// TIA Portal V20 export
FUNCTION_BLOCK "F-FB_DigitalInput"   // FB110, F_LAD
{ S7_Optimized_Access := 'TRUE' }
// stored: AutoNumber false
   VAR
      sSafety_EStop : EV1oo2DI;
      sKeySettingMode : EV1oo2DI;
      sKeySettingLaser : EV1oo2DI;
      sMaintenanceDoorClosed : EV1oo2DI;
      sFrontDoorClosed : EV1oo2DI;
      sEmergencyStopPowerLaser : EV1oo2DI;
      sRoofLeftDoorClosed : EV1oo2DI;
      sKeyLaserON : EV1oo2DI;
      sLaserExternDoorClosed : EV1oo2DI;
      sSasOneDoorClosed : EV1oo2DI;
      sBwLoaderDoorClosed : EV1oo2DI;
      sRoofRightDoorClosed : EV1oo2DI;
      sSonplas_EStop : EV1oo2DI;
      sBwLoader_EStop : EV1oo2DI;
      sSonplasDoorClosed : EV1oo2DI;
      sAck_iSafety_EStop { ExternalAccessible := 'False'; ExternalVisible := 'False'; ExternalWritable := 'False'} : Bool;
      sAck_iKeySettingMode { ExternalAccessible := 'False'; ExternalVisible := 'False'; ExternalWritable := 'False'} : Bool;
      sAck_iKeySettingLaser { ExternalAccessible := 'False'; ExternalVisible := 'False'; ExternalWritable := 'False'} : Bool;
      sAck_iMaintenanceDoorClosed { ExternalAccessible := 'False'; ExternalVisible := 'False'; ExternalWritable := 'False'} : Bool;
      sAck_iFrontDoorClosed { ExternalAccessible := 'False'; ExternalVisible := 'False'; ExternalWritable := 'False'} : Bool;
      sAck_iEmergencyStopPowerLaser { ExternalAccessible := 'False'; ExternalVisible := 'False'; ExternalWritable := 'False'} : Bool;
      sAck_iRoofLeftDoorClosed { ExternalAccessible := 'False'; ExternalVisible := 'False'; ExternalWritable := 'False'} : Bool;
      sAck_iKeyLaserON { ExternalAccessible := 'False'; ExternalVisible := 'False'; ExternalWritable := 'False'} : Bool;
      sAck_iLaserExternDoorClosed : Bool;
      sAck_iSasOneDoorClosed { ExternalAccessible := 'False'; ExternalVisible := 'False'; ExternalWritable := 'False'} : Bool;
      sAck_iBwLoaderDoorClosed : Bool;
      sAck_iRoofRightDoorClosed { ExternalAccessible := 'False'; ExternalVisible := 'False'; ExternalWritable := 'False'} : Bool;
      sAck_iSonplas_EStop : Bool;
      sAck_iBwLoader_EStop : Bool;
      sAck_iSonplasDoorClosed { ExternalAccessible := 'False'; ExternalVisible := 'False'; ExternalWritable := 'False'} : Bool;
   END_VAR
BEGIN

REGION Network 1: Safety EStop
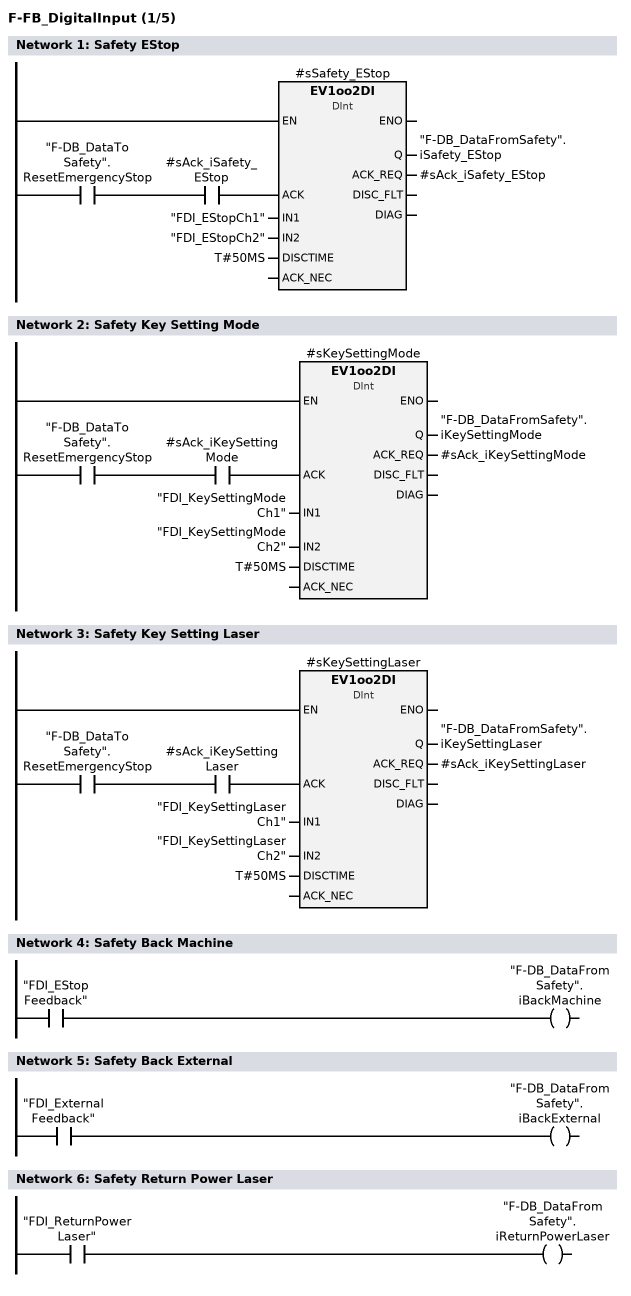
   RUNG wire#powerrail
      { S7_Templates := "codedbool_type := DInt" } #sSafety_EStop.EV1oo2DI(ACK := wire#w1, IN1 := "FDI_EStopCh1", IN2 := "FDI_EStopCh2", DISCTIME := T#50MS, ACK_NEC :=, Q => "F-DB_DataFromSafety".iSafety_EStop, ACK_REQ => #sAck_iSafety_EStop, DISC_FLT =>, DIAG =>)
   END_RUNG
   RUNG wire#powerrail
      Contact( "F-DB_DataToSafety".ResetEmergencyStop )
      Contact( #sAck_iSafety_EStop )
   END_RUNG wire#w1
   // the same network as SCL:
   #sSafety_EStop(ACK := "F-DB_DataToSafety".ResetEmergencyStop AND #sAck_iSafety_EStop,   // EV1oo2DI
                  IN1 := "FDI_EStopCh1",
                  IN2 := "FDI_EStopCh2",
                  DISCTIME := T#50MS,
                  Q => "F-DB_DataFromSafety".iSafety_EStop,
                  ACK_REQ => #sAck_iSafety_EStop);
END_REGION

REGION Network 2: Safety Key Setting Mode
   RUNG wire#powerrail
      { S7_Templates := "codedbool_type := DInt" } #sKeySettingMode.EV1oo2DI(ACK := wire#w1, IN1 := "FDI_KeySettingModeCh1", IN2 := "FDI_KeySettingModeCh2", DISCTIME := T#50MS, ACK_NEC :=, Q => "F-DB_DataFromSafety".iKeySettingMode, ACK_REQ => #sAck_iKeySettingMode, DISC_FLT =>, DIAG =>)
   END_RUNG
   RUNG wire#powerrail
      Contact( "F-DB_DataToSafety".ResetEmergencyStop )
      Contact( #sAck_iKeySettingMode )
   END_RUNG wire#w1
   // the same network as SCL:
   #sKeySettingMode(ACK := "F-DB_DataToSafety".ResetEmergencyStop AND #sAck_iKeySettingMode,   // EV1oo2DI
                    IN1 := "FDI_KeySettingModeCh1",
                    IN2 := "FDI_KeySettingModeCh2",
                    DISCTIME := T#50MS,
                    Q => "F-DB_DataFromSafety".iKeySettingMode,
                    ACK_REQ => #sAck_iKeySettingMode);
END_REGION

REGION Network 3: Safety Key Setting Laser
   RUNG wire#powerrail
      { S7_Templates := "codedbool_type := DInt" } #sKeySettingLaser.EV1oo2DI(ACK := wire#w1, IN1 := "FDI_KeySettingLaserCh1", IN2 := "FDI_KeySettingLaserCh2", DISCTIME := T#50MS, ACK_NEC :=, Q => "F-DB_DataFromSafety".iKeySettingLaser, ACK_REQ => #sAck_iKeySettingLaser, DISC_FLT =>, DIAG =>)
   END_RUNG
   RUNG wire#powerrail
      Contact( "F-DB_DataToSafety".ResetEmergencyStop )
      Contact( #sAck_iKeySettingLaser )
   END_RUNG wire#w1
   // the same network as SCL:
   #sKeySettingLaser(ACK := "F-DB_DataToSafety".ResetEmergencyStop AND #sAck_iKeySettingLaser,   // EV1oo2DI
                     IN1 := "FDI_KeySettingLaserCh1",
                     IN2 := "FDI_KeySettingLaserCh2",
                     DISCTIME := T#50MS,
                     Q => "F-DB_DataFromSafety".iKeySettingLaser,
                     ACK_REQ => #sAck_iKeySettingLaser);
END_REGION

REGION Network 4: Safety Back Machine
   RUNG wire#powerrail
      Contact( "FDI_EStopFeedback" )
      Coil( "F-DB_DataFromSafety".iBackMachine )
   END_RUNG
   // the same network as SCL:
   "F-DB_DataFromSafety".iBackMachine := "FDI_EStopFeedback";
END_REGION

REGION Network 5: Safety Back External
   RUNG wire#powerrail
      Contact( "FDI_ExternalFeedback" )
      Coil( "F-DB_DataFromSafety".iBackExternal )
   END_RUNG
   // the same network as SCL:
   "F-DB_DataFromSafety".iBackExternal := "FDI_ExternalFeedback";
END_REGION

REGION Network 6: Safety Return Power Laser
   RUNG wire#powerrail
      Contact( "FDI_ReturnPowerLaser" )
      Coil( "F-DB_DataFromSafety".iReturnPowerLaser )
   END_RUNG
   // the same network as SCL:
   "F-DB_DataFromSafety".iReturnPowerLaser := "FDI_ReturnPowerLaser";
END_REGION

REGION Network 7: Safety Maintenance Door Closed
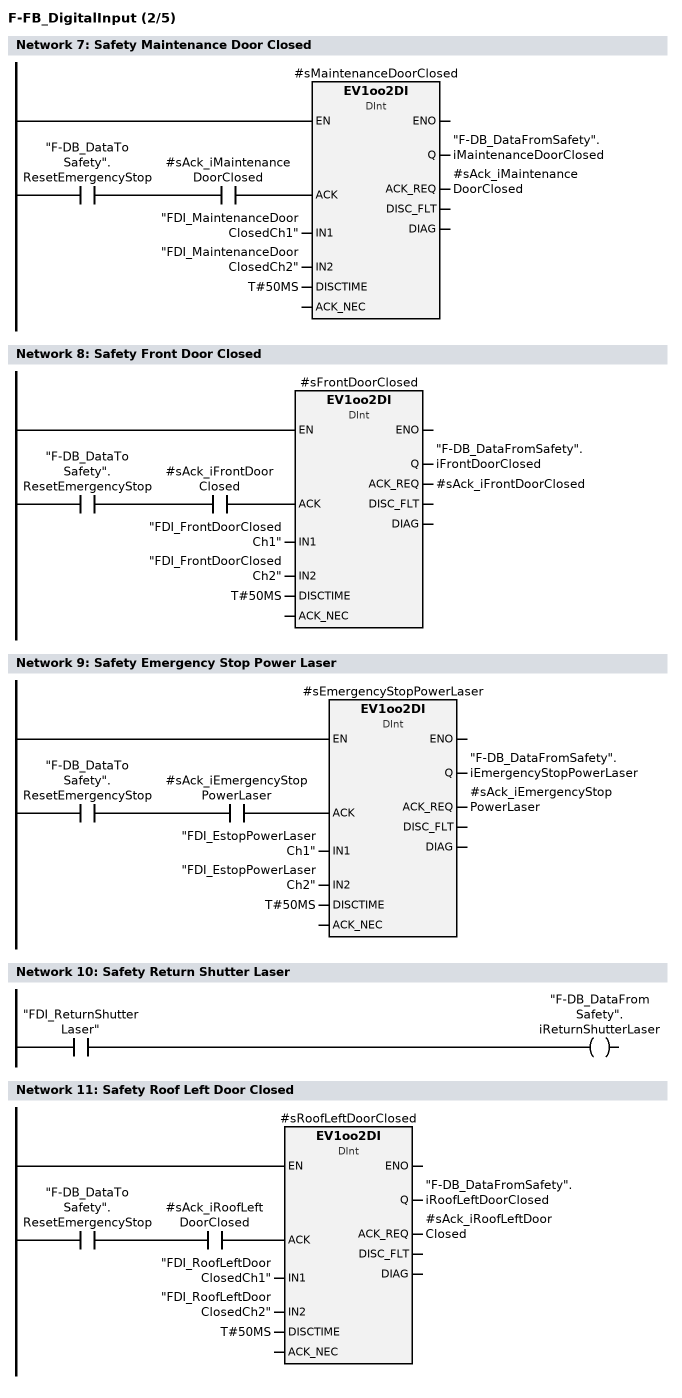
   RUNG wire#powerrail
      { S7_Templates := "codedbool_type := DInt" } #sMaintenanceDoorClosed.EV1oo2DI(ACK := wire#w1, IN1 := "FDI_MaintenanceDoorClosedCh1", IN2 := "FDI_MaintenanceDoorClosedCh2", DISCTIME := T#50MS, ACK_NEC :=, Q => "F-DB_DataFromSafety".iMaintenanceDoorClosed, ACK_REQ => #sAck_iMaintenanceDoorClosed, DISC_FLT =>, DIAG =>)
   END_RUNG
   RUNG wire#powerrail
      Contact( "F-DB_DataToSafety".ResetEmergencyStop )
      Contact( #sAck_iMaintenanceDoorClosed )
   END_RUNG wire#w1
   // the same network as SCL:
   #sMaintenanceDoorClosed(ACK := "F-DB_DataToSafety".ResetEmergencyStop AND #sAck_iMaintenanceDoorClosed,   // EV1oo2DI
                           IN1 := "FDI_MaintenanceDoorClosedCh1",
                           IN2 := "FDI_MaintenanceDoorClosedCh2",
                           DISCTIME := T#50MS,
                           Q => "F-DB_DataFromSafety".iMaintenanceDoorClosed,
                           ACK_REQ => #sAck_iMaintenanceDoorClosed);
END_REGION

REGION Network 8: Safety Front Door Closed
   RUNG wire#powerrail
      { S7_Templates := "codedbool_type := DInt" } #sFrontDoorClosed.EV1oo2DI(ACK := wire#w1, IN1 := "FDI_FrontDoorClosedCh1", IN2 := "FDI_FrontDoorClosedCh2", DISCTIME := T#50MS, ACK_NEC :=, Q => "F-DB_DataFromSafety".iFrontDoorClosed, ACK_REQ => #sAck_iFrontDoorClosed, DISC_FLT =>, DIAG =>)
   END_RUNG
   RUNG wire#powerrail
      Contact( "F-DB_DataToSafety".ResetEmergencyStop )
      Contact( #sAck_iFrontDoorClosed )
   END_RUNG wire#w1
   // the same network as SCL:
   #sFrontDoorClosed(ACK := "F-DB_DataToSafety".ResetEmergencyStop AND #sAck_iFrontDoorClosed,   // EV1oo2DI
                     IN1 := "FDI_FrontDoorClosedCh1",
                     IN2 := "FDI_FrontDoorClosedCh2",
                     DISCTIME := T#50MS,
                     Q => "F-DB_DataFromSafety".iFrontDoorClosed,
                     ACK_REQ => #sAck_iFrontDoorClosed);
END_REGION

REGION Network 9: Safety Emergency Stop Power Laser
   RUNG wire#powerrail
      { S7_Templates := "codedbool_type := DInt" } #sEmergencyStopPowerLaser.EV1oo2DI(ACK := wire#w1, IN1 := "FDI_EstopPowerLaserCh1", IN2 := "FDI_EstopPowerLaserCh2", DISCTIME := T#50MS, ACK_NEC :=, Q => "F-DB_DataFromSafety".iEmergencyStopPowerLaser, ACK_REQ => #sAck_iEmergencyStopPowerLaser, DISC_FLT =>, DIAG =>)
   END_RUNG
   RUNG wire#powerrail
      Contact( "F-DB_DataToSafety".ResetEmergencyStop )
      Contact( #sAck_iEmergencyStopPowerLaser )
   END_RUNG wire#w1
   // the same network as SCL:
   #sEmergencyStopPowerLaser(ACK := "F-DB_DataToSafety".ResetEmergencyStop AND #sAck_iEmergencyStopPowerLaser,   // EV1oo2DI
                           IN1 := "FDI_EstopPowerLaserCh1",
                           IN2 := "FDI_EstopPowerLaserCh2",
                           DISCTIME := T#50MS,
                           Q => "F-DB_DataFromSafety".iEmergencyStopPowerLaser,
                           ACK_REQ => #sAck_iEmergencyStopPowerLaser);
END_REGION

REGION Network 10: Safety Return Shutter Laser
   RUNG wire#powerrail
      Contact( "FDI_ReturnShutterLaser" )
      Coil( "F-DB_DataFromSafety".iReturnShutterLaser )
   END_RUNG
   // the same network as SCL:
   "F-DB_DataFromSafety".iReturnShutterLaser := "FDI_ReturnShutterLaser";
END_REGION

REGION Network 11: Safety Roof Left Door Closed
   RUNG wire#powerrail
      { S7_Templates := "codedbool_type := DInt" } #sRoofLeftDoorClosed.EV1oo2DI(ACK := wire#w1, IN1 := "FDI_RoofLeftDoorClosedCh1", IN2 := "FDI_RoofLeftDoorClosedCh2", DISCTIME := T#50MS, ACK_NEC :=, Q => "F-DB_DataFromSafety".iRoofLeftDoorClosed, ACK_REQ => #sAck_iRoofLeftDoorClosed, DISC_FLT =>, DIAG =>)
   END_RUNG
   RUNG wire#powerrail
      Contact( "F-DB_DataToSafety".ResetEmergencyStop )
      Contact( #sAck_iRoofLeftDoorClosed )
   END_RUNG wire#w1
   // the same network as SCL:
   #sRoofLeftDoorClosed(ACK := "F-DB_DataToSafety".ResetEmergencyStop AND #sAck_iRoofLeftDoorClosed,   // EV1oo2DI
                        IN1 := "FDI_RoofLeftDoorClosedCh1",
                        IN2 := "FDI_RoofLeftDoorClosedCh2",
                        DISCTIME := T#50MS,
                        Q => "F-DB_DataFromSafety".iRoofLeftDoorClosed,
                        ACK_REQ => #sAck_iRoofLeftDoorClosed);
END_REGION

REGION Network 12: Key Laser On
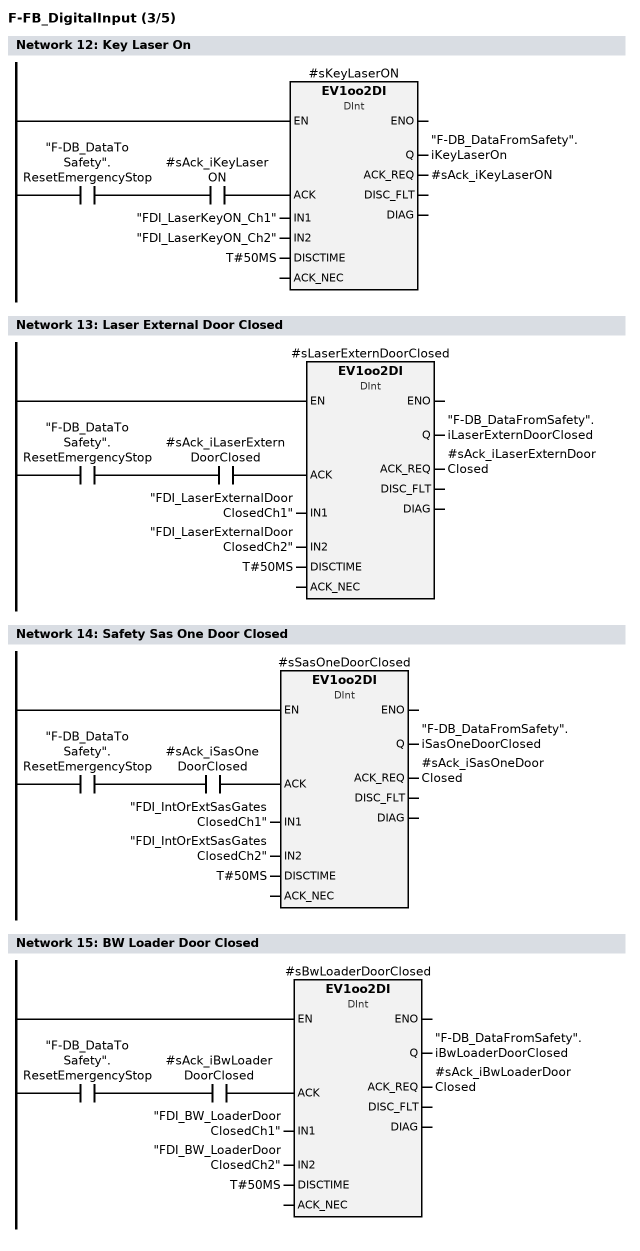
   RUNG wire#powerrail
      { S7_Templates := "codedbool_type := DInt" } #sKeyLaserON.EV1oo2DI(ACK := wire#w1, IN1 := "FDI_LaserKeyON_Ch1", IN2 := "FDI_LaserKeyON_Ch2", DISCTIME := T#50MS, ACK_NEC :=, Q => "F-DB_DataFromSafety".iKeyLaserOn, ACK_REQ => #sAck_iKeyLaserON, DISC_FLT =>, DIAG =>)
   END_RUNG
   RUNG wire#powerrail
      Contact( "F-DB_DataToSafety".ResetEmergencyStop )
      Contact( #sAck_iKeyLaserON )
   END_RUNG wire#w1
   // the same network as SCL:
   #sKeyLaserON(ACK := "F-DB_DataToSafety".ResetEmergencyStop AND #sAck_iKeyLaserON,   // EV1oo2DI
                IN1 := "FDI_LaserKeyON_Ch1",
                IN2 := "FDI_LaserKeyON_Ch2",
                DISCTIME := T#50MS,
                Q => "F-DB_DataFromSafety".iKeyLaserOn,
                ACK_REQ => #sAck_iKeyLaserON);
END_REGION

REGION Network 13: Laser External Door Closed
   RUNG wire#powerrail
      { S7_Templates := "codedbool_type := DInt" } #sLaserExternDoorClosed.EV1oo2DI(ACK := wire#w1, IN1 := "FDI_LaserExternalDoorClosedCh1", IN2 := "FDI_LaserExternalDoorClosedCh2", DISCTIME := T#50MS, ACK_NEC :=, Q => "F-DB_DataFromSafety".iLaserExternDoorClosed, ACK_REQ => #sAck_iLaserExternDoorClosed, DISC_FLT =>, DIAG =>)
   END_RUNG
   RUNG wire#powerrail
      Contact( "F-DB_DataToSafety".ResetEmergencyStop )
      Contact( #sAck_iLaserExternDoorClosed )
   END_RUNG wire#w1
   // the same network as SCL:
   #sLaserExternDoorClosed(ACK := "F-DB_DataToSafety".ResetEmergencyStop AND #sAck_iLaserExternDoorClosed,   // EV1oo2DI
                           IN1 := "FDI_LaserExternalDoorClosedCh1",
                           IN2 := "FDI_LaserExternalDoorClosedCh2",
                           DISCTIME := T#50MS,
                           Q => "F-DB_DataFromSafety".iLaserExternDoorClosed,
                           ACK_REQ => #sAck_iLaserExternDoorClosed);
END_REGION

REGION Network 14: Safety Sas One Door Closed
   RUNG wire#powerrail
      { S7_Templates := "codedbool_type := DInt" } #sSasOneDoorClosed.EV1oo2DI(ACK := wire#w1, IN1 := "FDI_IntOrExtSasGatesClosedCh1", IN2 := "FDI_IntOrExtSasGatesClosedCh2", DISCTIME := T#50MS, ACK_NEC :=, Q => "F-DB_DataFromSafety".iSasOneDoorClosed, ACK_REQ => #sAck_iSasOneDoorClosed, DISC_FLT =>, DIAG =>)
   END_RUNG
   RUNG wire#powerrail
      Contact( "F-DB_DataToSafety".ResetEmergencyStop )
      Contact( #sAck_iSasOneDoorClosed )
   END_RUNG wire#w1
   // the same network as SCL:
   #sSasOneDoorClosed(ACK := "F-DB_DataToSafety".ResetEmergencyStop AND #sAck_iSasOneDoorClosed,   // EV1oo2DI
                      IN1 := "FDI_IntOrExtSasGatesClosedCh1",
                      IN2 := "FDI_IntOrExtSasGatesClosedCh2",
                      DISCTIME := T#50MS,
                      Q => "F-DB_DataFromSafety".iSasOneDoorClosed,
                      ACK_REQ => #sAck_iSasOneDoorClosed);
END_REGION

REGION Network 15: BW Loader Door Closed
   RUNG wire#powerrail
      { S7_Templates := "codedbool_type := DInt" } #sBwLoaderDoorClosed.EV1oo2DI(ACK := wire#w1, IN1 := "FDI_BW_LoaderDoorClosedCh1", IN2 := "FDI_BW_LoaderDoorClosedCh2", DISCTIME := T#50MS, ACK_NEC :=, Q => "F-DB_DataFromSafety".iBwLoaderDoorClosed, ACK_REQ => #sAck_iBwLoaderDoorClosed, DISC_FLT =>, DIAG =>)
   END_RUNG
   RUNG wire#powerrail
      Contact( "F-DB_DataToSafety".ResetEmergencyStop )
      Contact( #sAck_iBwLoaderDoorClosed )
   END_RUNG wire#w1
   // the same network as SCL:
   #sBwLoaderDoorClosed(ACK := "F-DB_DataToSafety".ResetEmergencyStop AND #sAck_iBwLoaderDoorClosed,   // EV1oo2DI
                        IN1 := "FDI_BW_LoaderDoorClosedCh1",
                        IN2 := "FDI_BW_LoaderDoorClosedCh2",
                        DISCTIME := T#50MS,
                        Q => "F-DB_DataFromSafety".iBwLoaderDoorClosed,
                        ACK_REQ => #sAck_iBwLoaderDoorClosed);
END_REGION

REGION Network 16: Safety Right Door Closed
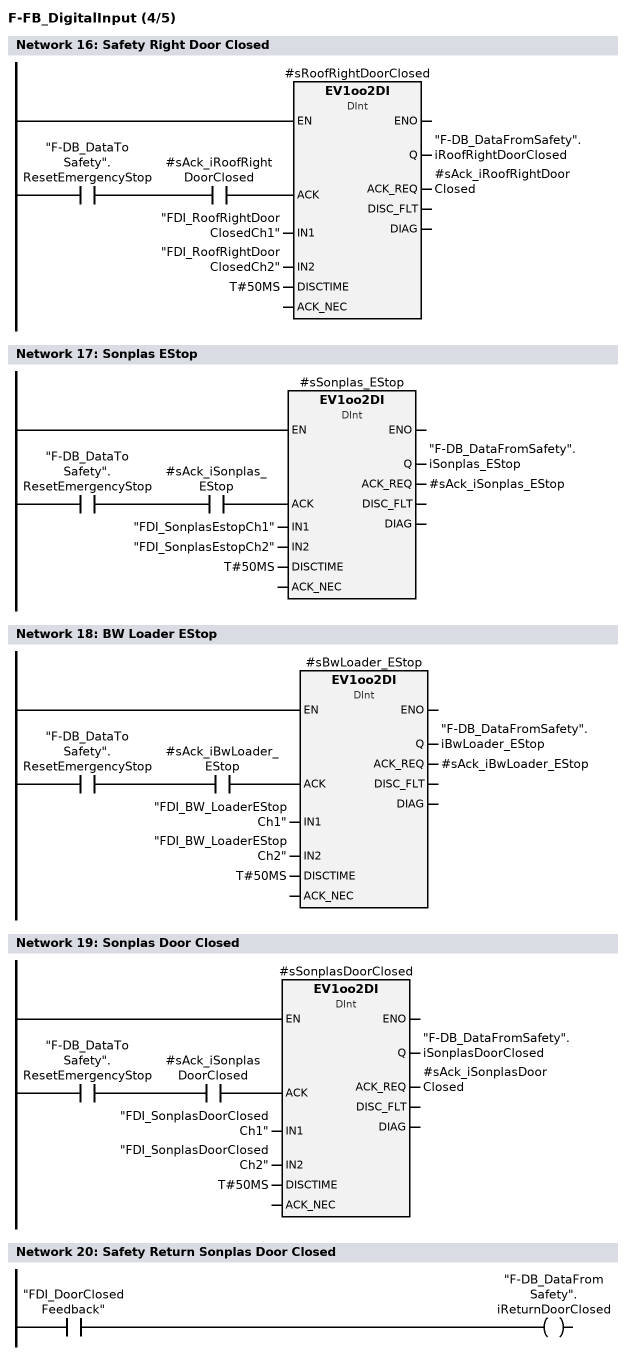
   RUNG wire#powerrail
      { S7_Templates := "codedbool_type := DInt" } #sRoofRightDoorClosed.EV1oo2DI(ACK := wire#w1, IN1 := "FDI_RoofRightDoorClosedCh1", IN2 := "FDI_RoofRightDoorClosedCh2", DISCTIME := T#50MS, ACK_NEC :=, Q => "F-DB_DataFromSafety".iRoofRightDoorClosed, ACK_REQ => #sAck_iRoofRightDoorClosed, DISC_FLT =>, DIAG =>)
   END_RUNG
   RUNG wire#powerrail
      Contact( "F-DB_DataToSafety".ResetEmergencyStop )
      Contact( #sAck_iRoofRightDoorClosed )
   END_RUNG wire#w1
   // the same network as SCL:
   #sRoofRightDoorClosed(ACK := "F-DB_DataToSafety".ResetEmergencyStop AND #sAck_iRoofRightDoorClosed,   // EV1oo2DI
                         IN1 := "FDI_RoofRightDoorClosedCh1",
                         IN2 := "FDI_RoofRightDoorClosedCh2",
                         DISCTIME := T#50MS,
                         Q => "F-DB_DataFromSafety".iRoofRightDoorClosed,
                         ACK_REQ => #sAck_iRoofRightDoorClosed);
END_REGION

REGION Network 17: Sonplas EStop
   RUNG wire#powerrail
      { S7_Templates := "codedbool_type := DInt" } #sSonplas_EStop.EV1oo2DI(ACK := wire#w1, IN1 := "FDI_SonplasEstopCh1", IN2 := "FDI_SonplasEstopCh2", DISCTIME := T#50MS, ACK_NEC :=, Q => "F-DB_DataFromSafety".iSonplas_EStop, ACK_REQ => #sAck_iSonplas_EStop, DISC_FLT =>, DIAG =>)
   END_RUNG
   RUNG wire#powerrail
      Contact( "F-DB_DataToSafety".ResetEmergencyStop )
      Contact( #sAck_iSonplas_EStop )
   END_RUNG wire#w1
   // the same network as SCL:
   #sSonplas_EStop(ACK := "F-DB_DataToSafety".ResetEmergencyStop AND #sAck_iSonplas_EStop,   // EV1oo2DI
                   IN1 := "FDI_SonplasEstopCh1",
                   IN2 := "FDI_SonplasEstopCh2",
                   DISCTIME := T#50MS,
                   Q => "F-DB_DataFromSafety".iSonplas_EStop,
                   ACK_REQ => #sAck_iSonplas_EStop);
END_REGION

REGION Network 18: BW Loader EStop
   RUNG wire#powerrail
      { S7_Templates := "codedbool_type := DInt" } #sBwLoader_EStop.EV1oo2DI(ACK := wire#w1, IN1 := "FDI_BW_LoaderEStopCh1", IN2 := "FDI_BW_LoaderEStopCh2", DISCTIME := T#50MS, ACK_NEC :=, Q => "F-DB_DataFromSafety".iBwLoader_EStop, ACK_REQ => #sAck_iBwLoader_EStop, DISC_FLT =>, DIAG =>)
   END_RUNG
   RUNG wire#powerrail
      Contact( "F-DB_DataToSafety".ResetEmergencyStop )
      Contact( #sAck_iBwLoader_EStop )
   END_RUNG wire#w1
   // the same network as SCL:
   #sBwLoader_EStop(ACK := "F-DB_DataToSafety".ResetEmergencyStop AND #sAck_iBwLoader_EStop,   // EV1oo2DI
                    IN1 := "FDI_BW_LoaderEStopCh1",
                    IN2 := "FDI_BW_LoaderEStopCh2",
                    DISCTIME := T#50MS,
                    Q => "F-DB_DataFromSafety".iBwLoader_EStop,
                    ACK_REQ => #sAck_iBwLoader_EStop);
END_REGION

REGION Network 19: Sonplas Door Closed
   RUNG wire#powerrail
      { S7_Templates := "codedbool_type := DInt" } #sSonplasDoorClosed.EV1oo2DI(ACK := wire#w1, IN1 := "FDI_SonplasDoorClosedCh1", IN2 := "FDI_SonplasDoorClosedCh2", DISCTIME := T#50MS, ACK_NEC :=, Q => "F-DB_DataFromSafety".iSonplasDoorClosed, ACK_REQ => #sAck_iSonplasDoorClosed, DISC_FLT =>, DIAG =>)
   END_RUNG
   RUNG wire#powerrail
      Contact( "F-DB_DataToSafety".ResetEmergencyStop )
      Contact( #sAck_iSonplasDoorClosed )
   END_RUNG wire#w1
   // the same network as SCL:
   #sSonplasDoorClosed(ACK := "F-DB_DataToSafety".ResetEmergencyStop AND #sAck_iSonplasDoorClosed,   // EV1oo2DI
                       IN1 := "FDI_SonplasDoorClosedCh1",
                       IN2 := "FDI_SonplasDoorClosedCh2",
                       DISCTIME := T#50MS,
                       Q => "F-DB_DataFromSafety".iSonplasDoorClosed,
                       ACK_REQ => #sAck_iSonplasDoorClosed);
END_REGION

REGION Network 20: Safety Return Sonplas Door Closed
   RUNG wire#powerrail
      Contact( "FDI_DoorClosedFeedback" )
      Coil( "F-DB_DataFromSafety".iReturnDoorClosed )
   END_RUNG
   // the same network as SCL:
   "F-DB_DataFromSafety".iReturnDoorClosed := "FDI_DoorClosedFeedback";
END_REGION

REGION Network 21: Manage Acknowledge Request
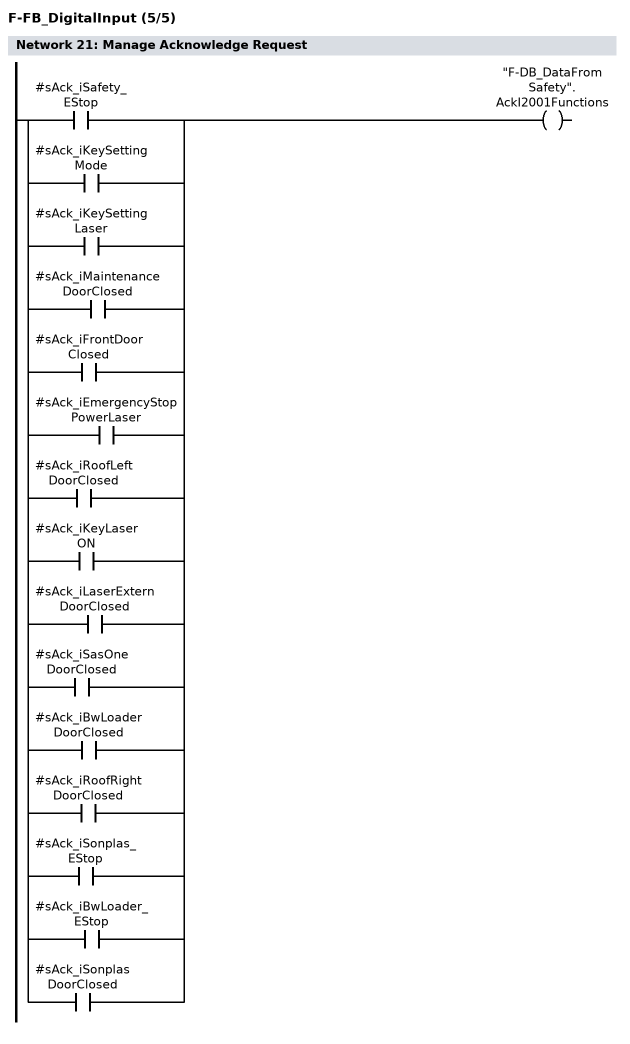
   RUNG wire#powerrail
      Contact( #sAck_iSafety_EStop )
      wire#w1
      Coil( "F-DB_DataFromSafety".AckI2001Functions )
   END_RUNG
   RUNG wire#powerrail
      Contact( #sAck_iKeySettingMode )
   END_RUNG wire#w1
   RUNG wire#powerrail
      Contact( #sAck_iKeySettingLaser )
   END_RUNG wire#w1
   RUNG wire#powerrail
      Contact( #sAck_iMaintenanceDoorClosed )
   END_RUNG wire#w1
   RUNG wire#powerrail
      Contact( #sAck_iFrontDoorClosed )
   END_RUNG wire#w1
   RUNG wire#powerrail
      Contact( #sAck_iEmergencyStopPowerLaser )
   END_RUNG wire#w1
   RUNG wire#powerrail
      Contact( #sAck_iRoofLeftDoorClosed )
   END_RUNG wire#w1
   RUNG wire#powerrail
      Contact( #sAck_iKeyLaserON )
   END_RUNG wire#w1
   RUNG wire#powerrail
      Contact( #sAck_iLaserExternDoorClosed )
   END_RUNG wire#w1
   RUNG wire#powerrail
      Contact( #sAck_iSasOneDoorClosed )
   END_RUNG wire#w1
   RUNG wire#powerrail
      Contact( #sAck_iBwLoaderDoorClosed )
   END_RUNG wire#w1
   RUNG wire#powerrail
      Contact( #sAck_iRoofRightDoorClosed )
   END_RUNG wire#w1
   RUNG wire#powerrail
      Contact( #sAck_iSonplas_EStop )
   END_RUNG wire#w1
   RUNG wire#powerrail
      Contact( #sAck_iBwLoader_EStop )
   END_RUNG wire#w1
   RUNG wire#powerrail
      Contact( #sAck_iSonplasDoorClosed )
   END_RUNG wire#w1
   // the same network as SCL:
   "F-DB_DataFromSafety".AckI2001Functions := #sAck_iSafety_EStop OR #sAck_iKeySettingMode OR #sAck_iKeySettingLaser OR #sAck_iMaintenanceDoorClosed OR #sAck_iFrontDoorClosed OR #sAck_iEmergencyStopPowerLaser OR #sAck_iRoofLeftDoorClosed OR #sAck_iKeyLaserON OR #sAck_iLaserExternDoorClosed OR #sAck_iSasOneDoorClosed OR #sAck_iBwLoaderDoorClosed OR #sAck_iRoofRightDoorClosed OR #sAck_iSonplas_EStop OR #sAck_iBwLoader_EStop OR #sAck_iSonplasDoorClosed;
END_REGION
END_FUNCTION_BLOCK
